// LS Electric XG5000 project: 과년68_2_3
// PLC NewPLC
// module base 0 slot 0: 입출력 모듈:XBC-DR20S (DC 24V 입력 12점, 릴레이 출력 8점)

PROGRAM NewProgram (task: 스캔 프로그램)

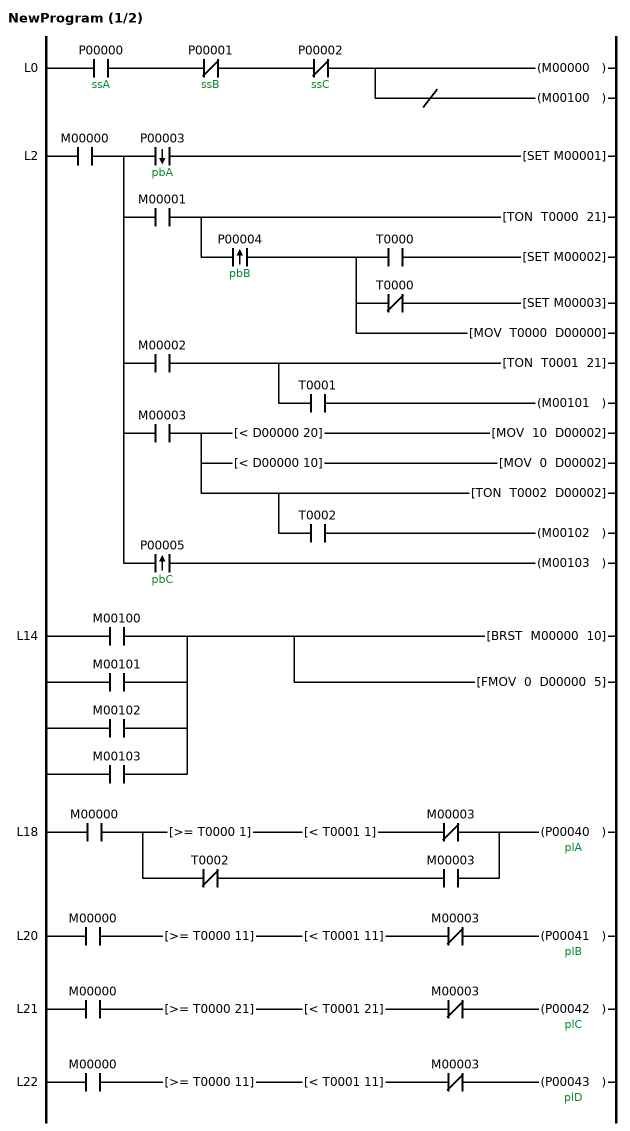
; L0
LOAD      P00000	// ssA
AND NOT   P00001	// ssB
AND NOT   P00002	// ssC
OUT       M00000
NOT
OUT       M00100
; L2
LOAD      M00000
MPUSH
ANDN      P00003	// pbA
SET       M00001
MLOAD
AND       M00001
TON       T0000 21
ANDP      P00004	// pbB
MPUSH
AND       T0000
SET       M00002
MLOAD
AND NOT   T0000
SET       M00003
MPOP
MOV       T0000 D00000
MLOAD
AND       M00002
TON       T0001 21
AND       T0001
OUT       M00101
MLOAD
AND       M00003
MPUSH
AND<      D00000 20
MOV       10 D00002
MLOAD
AND<      D00000 10
MOV       0 D00002
MPOP
TON       T0002 D00002
AND       T0002
OUT       M00102
MPOP
ANDP      P00005	// pbC
OUT       M00103
; L14
LOAD      M00100
OR        M00101
OR        M00102
OR        M00103
BRST      M00000 10
FMOV      0 D00000 5
; L18
LOAD      M00000
LOAD>=    T0000 1
AND<      T0001 1
AND NOT   M00003
LOAD NOT  T0002
AND       M00003
OR LOAD
AND LOAD
OUT       P00040	// plA
; L20
LOAD      M00000
AND>=     T0000 11
AND<      T0001 11
AND NOT   M00003
OUT       P00041	// plB
; L21
LOAD      M00000
AND>=     T0000 21
AND<      T0001 21
AND NOT   M00003
OUT       P00042	// plC
; L22
LOAD      M00000
AND>=     T0000 11
AND<      T0001 11
AND NOT   M00003
OUT       P00043	// plD

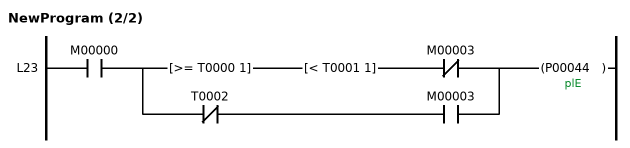
; L23
LOAD      M00000
LOAD>=    T0000 1
AND<      T0001 1
AND NOT   M00003
LOAD NOT  T0002
AND       M00003
OR LOAD
AND LOAD
OUT       P00044	// plE